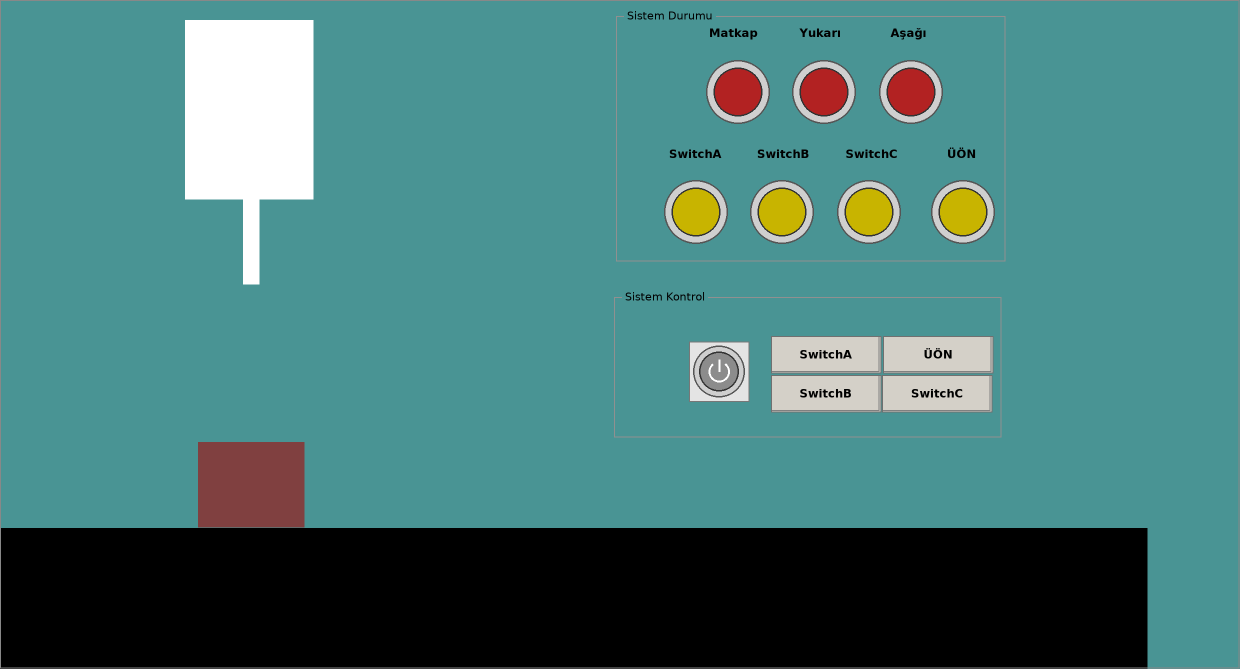
VISUALIZATION Visualization  // 1240x669
    Rectangle (-93,528 1240x141)
    Rectangle (198,442 106x85), invisible if: MAIN.C
    Group (185,20 128x264)
        p2738717112: MAIN.fDrillY
        Rectangle (58,164 16x100)
        Rectangle (0,0 128x179)
    Lamp1 (699,55 78x74), variable: MAIN.Drill.OUT.bDrill, style: Lamp-Lamp1-Red
    Lamp1 (785,55 78x74), variable: MAIN.Drill.OUT.bUp, style: Lamp-Lamp1-Red
    Lamp1 (872,55 78x74), variable: MAIN.Drill.OUT.bDown, style: Lamp-Lamp1-Red
    Label (702,18 63x30), "Matkap"
    Label (789,18 63x30), "Yukarı"
    Label (877,18 63x30), "Aşağı"
    Lamp1 (657,175 78x74), variable: MAIN.Drill.IN.bSwitchA, style: Lamp-Lamp1-Yellow
    Lamp1 (743,175 78x74), variable: MAIN.Drill.IN.bSwitchB, style: Lamp-Lamp1-Yellow
    Lamp1 (830,175 78x74), variable: MAIN.Drill.IN.bSwitchC, style: Lamp-Lamp1-Yellow
    Lamp1 (924,175 78x74), variable: MAIN.Drill.IN.bUpSwitch, style: Lamp-Lamp1-Yellow
    Label (664,139 63x30), "SwitchA"
    Label (752,139 63x30), "SwitchB"
    Label (840,139 63x30), "SwitchC"
    Label (930,139 63x30), "ÜÖN"
    Button (771,336 110x37), "SwitchA"
        toggle MAIN.Drill.IN.bSwitchA
    Button (771,375 110x37), "SwitchB"
        toggle MAIN.Drill.IN.bSwitchB
    Button (882,375 110x37), "SwitchC"
        toggle MAIN.Drill.IN.bSwitchC
    Button (883,336 110x37), "ÜÖN"
        toggle MAIN.Drill.IN.bUpSwitch
    PowerSwitch (689,341 60x61), variable: MAIN.Drill.IN.bStart, behaviour: TOGGLE, style: Switch-PowerSwitch-Gray
    GroupBox (616,8 389x253), "Sistem Durumu"
    GroupBox (614,289 387x148), "Sistem Kontrol"
END_VISUALIZATION

(* stored: Version 1.1.0.1, ProductVersion 3.1.4024.4
   Visu Visualization: Id {1b29ddf4-5f3e-4f69-ae2e-01779d835f33} *)
